(* Logix 5000 project; controller ASTEST_COUNTER_LAB 1769-L16ER-BB1B rev 32.15; software revision 32.05 *)

TASK MainTask (continuous, watchdog 500 ms) : MainProgram

MODULES
   Local : 1769-L16ER-BB1B (PointIO 0, rev 32.15)
      Discrete_IO : Embedded (PointIO 1, rev 32.11, Output RPI 20 ms)
           Local:1:O.Data.0   // RED
           Local:1:O.Data.1   // GREEN
           Local:1:O.Data.2   // BLUE
           Local:1:O.Data.3   // YELLOW
END_MODULES

PROGRAM MainProgram   (* main routine MainRoutine *)
VAR
   blink : DINT;
   blink1 : TIMER := (PRE := 1000, ACC := 1000, EN := 1, DN := 1);
   blink2 : TIMER := (PRE := 1000, ACC := 466, EN := 1, TT := 1);
   blinkBOOL : BOOL := 1;
   COUNTER : COUNTER := (ACC := 2, CD := 1, DN := 1);
        .PRE   // Keeps the counter in the DONE or NOT Done state
   interval : DINT := 8;
   START : BOOL := 1;
   TON : TIMER := (PRE := 10000, ACC := 8319, EN := 1, TT := 1);
END_VAR

ROUTINE MainRoutine   (* ladder *)
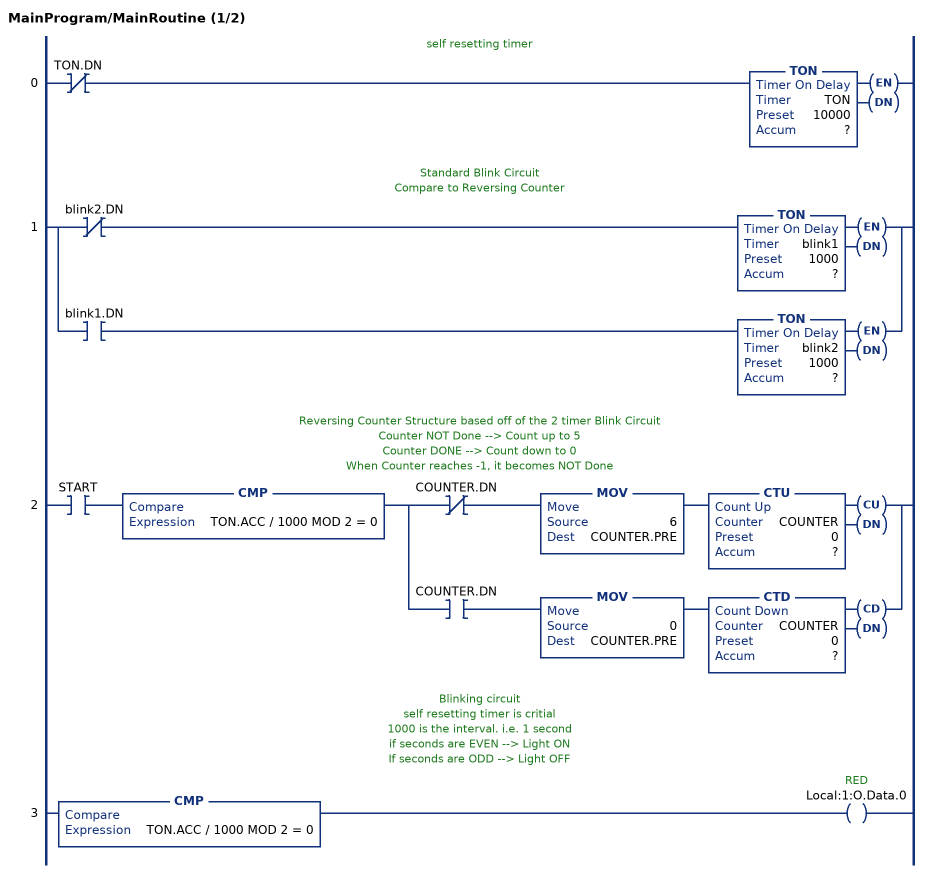
   // self resetting timer
   0: XIO(TON.DN)TON(TON,?,?);
   // Standard Blink Circuit
   // Compare to Reversing Counter
   1: [XIO(blink2.DN) TON(blink1,?,?) ,XIC(blink1.DN) TON(blink2,?,?) ];
   // Reversing Counter Structure based off of the 2 timer Blink Circuit
   // Counter NOT Done --> Count up to 5
   // Counter DONE --> Count down to 0
   // When Counter reaches -1, it becomes NOT Done
   2: XIC(START)CMP(TON.ACC / 1000 MOD 2 = 0)[XIO(COUNTER.DN) MOV(6,COUNTER.PRE) CTU(COUNTER,?,?) ,XIC(COUNTER.DN) MOV(0,COUNTER.PRE) CTD(COUNTER,?,?) ];
   // Blinking circuit
   // self resetting timer is critial
   // 1000 is the interval. i.e. 1 second
   // if seconds are EVEN --> Light ON
   // If seconds are ODD --> Light OFF
   3: CMP(TON.ACC / 1000 MOD 2 = 0)OTE(Local:1:O.Data.0);
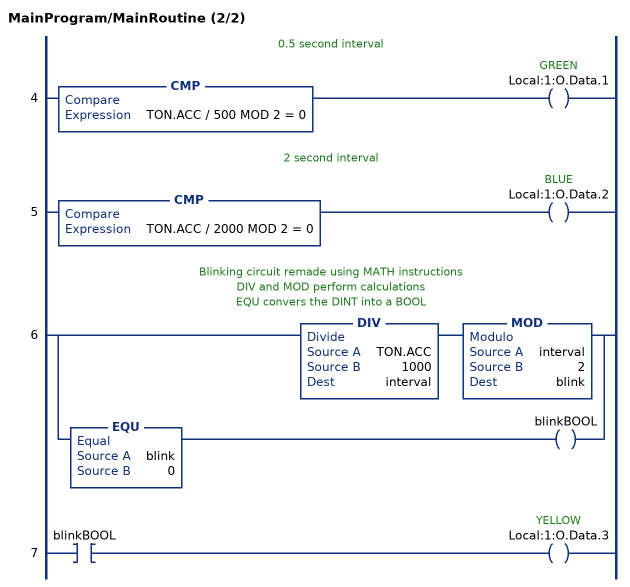
   // 0.5 second interval
   4: CMP(TON.ACC / 500 MOD 2 = 0)OTE(Local:1:O.Data.1);
   // 2 second interval
   5: CMP(TON.ACC / 2000 MOD 2 = 0)OTE(Local:1:O.Data.2);
   // Blinking circuit remade using MATH instructions
   // DIV and MOD perform calculations
   // EQU convers the DINT into a BOOL
   6: [DIV(TON.ACC,1000,interval) MOD(interval,2,blink) ,EQU(blink,0) OTE(blinkBOOL) ];
   7: XIC(blinkBOOL)OTE(Local:1:O.Data.3);
END_ROUTINE
END_PROGRAM
